{attribute addProperty BoxType "AT2026-0250-0019"}
{attribute addProperty Id "A_0077_AT2001_5250_0018_AT2001_5250AT2001_3DCFC8D064080"}
{attribute addProperty CRC "2912964423"}
{attribute addProperty SizeInBites "640"}
{attribute addProperty SizeInBytes "80"}
TYPE A_0065_AT2026_0250_0019_AT2026_0250_ADA04F47 EXTENDS AT2026_9506A482 :
STRUCT
	{attribute addProperty Name "A_0077_AT2001_5250_0018_AT2001_5250"}
	A_0077_AT2001_5250_0018_AT2001_5250 : AT2001_3DCFC8D0;
END_STRUCT
END_TYPE

(* stored: Version 1.2.0.0, ProductVersion 3.1.4024.9
   DUT A_0065_AT2026_0250_0019_AT2026_0250_ADA04F47: Id {3547c08d-6ca7-4d56-981f-77e771f1e0b9} *)
